{attribute 'qualified_only'}
{attribute 'strict'}
TYPE E_RestorePosition :
(
    eDontRestore :=0,
    eRestoreWithoutHome := 1 //Redefined the position of the axis to that when the power was lost
);
END_TYPE

(* stored: Version 1.1.0.1, ProductVersion 3.1.4024.5
   DUT E_RestorePosition: Id {74fe66e5-f3db-4a55-9501-11365c4561a4} *)
